// TIA Portal V19 export
VAR_GLOBAL   // PLC tag table "sys"
   Clock_Byte AT %MB0 : Byte;
   Clock_10Hz AT %M0.0 : Bool;
   Clock_5Hz AT %M0.1 : Bool;
   "Clock_2.5Hz" AT %M0.2 : Bool;
   Clock_2Hz AT %M0.3 : Bool;
   "Clock_1.25Hz" AT %M0.4 : Bool;
   Clock_1Hz AT %M0.5 : Bool;
   "Clock_0.625Hz" AT %M0.6 : Bool;
   "Clock_0.5Hz" AT %M0.7 : Bool;
   System_Byte AT %MB1 : Byte;
   FirstScan AT %M1.0 : Bool;
   DiagStatusUpdate AT %M1.1 : Bool;
   "TIME: 0.1sec" AT %M2.0 : Bool;
   "TIME: 0.2sec" AT %M2.1 : Bool;
   "TIME: 0.4sec" AT %M2.2 : Bool;
   "TIME: 0.5sec" AT %M2.3 : Bool;
   "TIME: 0.8sec" AT %M2.4 : Bool;
   "TIME: 1.0sec" AT %M2.5 : Bool;
   "TIME: 1.6sec" AT %M2.6 : Bool;
   "TIME: 2.0sec" AT %M2.7 : Bool;
   p1s AT %M20.0 : Bool;
   p100ms AT %M20.1 : Bool;
   ManualSET AT %M20.3 : Bool;
   AutoSET AT %M20.4 : Bool;
   generalAckn AT %M21.1 : Bool;
   AcknFaults AT %M21.2 : Bool;
   MuteHorn AT %M21.3 : Bool;
   ResetFaults AT %M21.4 : Bool;
   blink AT %M20.2 : Bool;
   RemAcknFaults AT %M21.5 : Bool;
   RemMuteSiren AT %M21.6 : Bool;
   RemResetFaults AT %M21.7 : Bool;
   Time_Byte AT %MB2 : Byte;
   "TIME: 0.1sec_OB30" AT %M4.0 : Bool;   // TIME: 100ms counted in cyclic OB30
   "TIME: 1.0sec_OB30" AT %M4.1 : Bool;   // TIME: 1s counted in cyclic OB30
   TIMECOUNTER_OB30 AT %MW8 : Int;
   Clock_1Hz_OB30 AT %M4.2 : Bool;   // CLOCK: 1s on / 1s off in cyclic OB30
   AlwaysTRUE AT %M1.2 : Bool;
   AlwaysFALSE AT %M1.3 : Bool;
END_VAR
